Staubli VAL3: nDialogInsNum.pgx

public program nDialogInsNum(string x_sTitle, string x_sText_r1, num& x_nNum)
  local num l_nVal
  local num l_nKey
begin

  //notes: screen size is 13rowsX40columns
  //usage: call DialogInsNums("NUMERIC INS", "Insert a value for foo:", num, screen)

  wait(getKey()==-1)
  userPage()
  call clrscr()
  l_nVal=x_nNum


  call sCenterTitle(x_sTitle)

  title(x_sTitle)

  gotoxy(0,4)
  //call sCenterRow(x_sText_r1)
  put(x_sText_r1)

  gotoxy(34,13)
  put("F8=Ok")

  gotoxy(0,13)
  put("F1=Esc")

  gotoxy(len(x_sText_r1)+1,4)
  gotoxy(len(x_sText_r1)+1, 4)


  do
    l_nKey=get(l_nVal)
    if l_nKey==278
      x_nNum=l_nVal
    endIf
  until l_nKey==271 or l_nKey==278

  call clrscr()
  wait(getKey()==-1)

end
